screen "04_Izleme" 800x480, template "MainTemplate"
   TextField "Text field_1" at 81,3 size 108x20; Text 'En Ayar Pistonu'
   TextField "Text field_2" at 139,27 size 51x20; Text 'İleride'
   Circle "Circle_1" at 148,52 size 34x34
      Appearance <- "Peripheral_Data_IN_EnAyar_P1_Ileride"
   TextField "Text field_3" at 200,27 size 51x20; Text 'Geride'
   Circle "Circle_2" at 209,52 size 34x34
      Appearance <- "Peripheral_Data_IN_EnAyar_P1_Geride"
   Circle "Circle_3" at 148,96 size 34x34
      Appearance <- "Peripheral_Data_IN_EnAyar_P2_Ileride"
   Circle "Circle_4" at 209,96 size 34x34
      Appearance <- "Peripheral_Data_IN_EnAyar_P2_Geride"
   TextField "Text field_4" at 42,60 size 60x20; Text 'P1 (sol):'
   TextField "Text field_5" at 43,101 size 65x20; Text 'P2 (sağ):'
   Circle "Circle_5" at 148,138 size 34x34
      Appearance <- "Peripheral_Data_IN_EnAyar_P1A_Ileride"
   Circle "Circle_6" at 209,138 size 34x34
      Appearance <- "Peripheral_Data_IN_EnAyar_P1A_Geride"
   Circle "Circle_7" at 148,182 size 34x34
      Appearance <- "Peripheral_Data_IN_EnAyar_P2A_Ileride"
   Circle "Circle_8" at 209,182 size 34x34
      Appearance <- "Peripheral_Data_IN_EnAyar_P2A_Geride"
   TextField "Text field_6" at 42,146 size 70x20; Text 'P1A (sol):'
   TextField "Text field_7" at 43,187 size 75x20; Text 'P2A (sağ):'
   TextField "Text field_8" at 606,3 size 108x20; Text 'Kademe Pistonu'
   TextField "Text field_9" at 664,27 size 51x20; Text 'İleride'
   Circle "Circle_9" at 673,52 size 34x34
      Appearance <- "Peripheral_Data_IN_KademeAyar_P3_Ileride"
   TextField "Text field_10" at 725,27 size 51x20; Text 'Geride'
   Circle "Circle_10" at 734,52 size 34x34
      Appearance <- "Peripheral_Data_IN_KademeAyar_P3_Geride"
   TextField "Text field_11" at 567,60 size 26x20; Text 'P3:'
   TextField "Text field_13" at 318,2 size 155x20; Text 'Kenetleme Pistonu'
   TextField "Text field_14" at 401,26 size 51x20; Text 'İleride'
   Circle "Circle_13" at 410,51 size 34x34
      Appearance <- "Peripheral_Data_IN_Kenetleme_P4_Ilderide"
   TextField "Text field_15" at 462,26 size 51x20; Text 'Geride'
   Circle "Circle_14" at 471,51 size 34x34
      Appearance <- "Peripheral_Data_IN_Kenetleme_P4_Geride"
   TextField "Text field_16" at 304,59 size 65x20; Text 'P4 (sağ):'
   Circle "Circle_17" at 410,96 size 34x34
      Appearance <- "Peripheral_Data_IN_Kenetleme_P4B_Ilderide"
   Circle "Circle_18" at 471,96 size 34x34
      Appearance <- "Peripheral_Data_IN_Kenetleme_P4B_Geride"
   TextField "Text field_18" at 304,104 size 68x20; Text 'P4B (sol):'
   TextField "Text field_20" at 81,231 size 108x20; Text 'İkaz Lambaları'
   Circle "Circle_21" at 178,260 size 34x34
      Appearance <- "Peripheral_Data_OUT_LAMBA_Yesil"
   TextField "Text field_23" at 42,268 size 40x20; Text 'Yeşil:'
   TextField "Text field_21" at 322,231 size 155x20; Text 'Diğer Ekipmanlar'
   Circle "Circle_22" at 441,261 size 34x34
      Appearance <- "Peripheral_Data_OUT_VacumJeneratoru"
   TextField "Text field_22" at 304,268 size 53x20; Text 'Vakum:'
   Circle "Circle_24" at 441,305 size 34x34
      Appearance <- "Peripheral_Data_OUT_VincLambasi"
   TextField "Text field_25" at 304,311 size 93x20; Text 'Vinc Lambası:'
   Circle "Circle_25" at 177,305 size 34x34
      Appearance <- "Peripheral_Data.OUT.LAMBA.Sari"
   TextField "Text field_26" at 42,310 size 35x20; Text 'Sarı:'
   Circle "Circle_11" at 440,351 size 34x34
      Appearance <- "Peripheral_Data.OUT.LAMBA.Buzzer"
   TextField "Text field_12" at 305,356 size 43x20; Text 'Siren:'
   Circle "Circle_23" at 178,351 size 34x34
      Appearance <- "Peripheral_Data_OUT_LAMBA_Kirmizi"
   TextField "Text field_24" at 43,356 size 51x20; Text 'Kırmızı:'
   TextField "Text field_17" at 149,59 size 30x20; Text 'I0.4'
   TextField "Text field_19" at 212,59 size 30x20; Text 'I0.5'
   TextField "Text field_27" at 149,103 size 30x20; Text 'I1.0'
   TextField "Text field_28" at 212,103 size 30x20; Text 'I1.1'
   TextField "Text field_29" at 149,145 size 30x20; Text 'I0.6'
   TextField "Text field_30" at 212,145 size 30x20; Text 'I0.7'
   TextField "Text field_31" at 149,189 size 30x20; Text 'I1.2'
   TextField "Text field_32" at 212,189 size 30x20; Text 'I1.3'
   TextField "Text field_33" at 411,57 size 30x20; Text 'I2.0'
   TextField "Text field_34" at 474,57 size 30x20; Text 'I2.1'
   TextField "Text field_35" at 412,102 size 30x20; Text 'I2.2'
   TextField "Text field_36" at 474,102 size 30x20; Text 'I2.3'
   TextField "Text field_37" at 674,59 size 30x20; Text 'I1.4'
   TextField "Text field_38" at 737,59 size 30x20; Text 'I1.5'
   TextField "Text field_39" at 178,267 size 34x20; Text 'Q0.2'
   TextField "Text field_40" at 178,311 size 34x20; Text 'Q0.1'
   TextField "Text field_41" at 178,357 size 34x20; Text 'Q0.0'
   TextField "Text field_42" at 440,267 size 34x20; Text 'Q0.3'
   TextField "Text field_43" at 440,310 size 34x20; Text 'Q0.4'
   TextField "Text field_44" at 440,357 size 34x20; Text 'Q0.5'

screen "05_Receipt" 800x480, template "MainTemplate"
   TextField "Text field_1" at 258,159 size 300x124; Text 'KAYDEDİLDİ'
      Visibility <- "Receipt_bShowMessage"
   TextField "Template_Text field_1" at 45,17 size 109x22; Text 'Model Seçimi:'
   SymbolicIOField "Template_Symbolic I/O field_1" at 270,13 size 524x32; TextOn '1'; TextOff '0'; TextList "textListReceipt"
      ProcessValue <- "ModelId"
   Button "btnSave" at 619,337 size 167x58; TextOff 'KAYDET'
      on Release: SetBit("Receipt_btnSave")
   TextField "Template_Text field_4" at 45,139 size 124x22; Text 'Model Boyu (C):'
   TextField "Template_Text field_2" at 46,57 size 83x22; Text 'Model Adı:'
   IOField "I/O field_1" at 274,53 size 524x32; FormatPattern ??????????????????????????????????????????????????
      ProcessValue <- "ModelName"
   IOField "I/O field_2" at 273,134 size 256x32; FormatPattern s9999999.99; Unit  mm
      ProcessValue <- "Receipt_CurrentModel_Boy_C"
   TextField "Template_Text field_5" at 46,181 size 111x22; Text 'Model Eni (D):'
   IOField "I/O field_3" at 274,175 size 256x32; FormatPattern s9999999.99; Unit  mm
      ProcessValue <- "Receipt_CurrentModel_En_D"
   TextField "Template_Text field_3" at 45,98 size 99x22; Text 'Model Sınıfı:'
   SymbolicIOField "Template_Symbolic I/O field_2" at 275,94 size 68x32; TextOn '1'; TextOff '0'; TextList "classList"
      ProcessValue <- "Receipt_CurrentModel_Class"
   IOField "I/O field_4" at 275,290 size 185x32; FormatPattern 99999.99; Unit  mm
      ProcessValue <- "HMI_Data_ServoData_txtGerdirmeMes"
   TextField "Template_Text field_6" at 46,294 size 151x22; Text 'Gerdirme Mesafesi:'
   TextField "Template_Text field_7" at 45,252 size 154x23; Text 'Kenetleme Süresi:'
   IOField "Template_I/O field_1" at 275,248 size 184x32; FormatPattern 9999999999; Unit  sn
      ProcessValue <- "HMI_Data_KenetlemeSuresi"

screen "06_Alarm" 800x480, template "MainTemplate"
   AlarmView "Alarm view_1" at 2,1 size 796x415

screen "Screen_1" 800x480
   TextField "Text field_4" at 293,58 size 227x20; Text 'SERVO OTOMATİK KONTROL'
   IOField "I/O field_4" at 304,101 size 202x39; FormatPattern 999.9; Unit  %
      ProcessValue <- "HMI_Data_ServoData_txtVelocity"
   TextField "Text field_6" at 74,110 size 134x20; Text 'OTOMATİK MOD HIZ:'
   Button "btnIncJogSpeedXaxis_1" at 224,102 size 74x37; TextOff '-'
      on Release: function_b9b71300("HMI_Data_ServoData_txtVelocity", 5)
   Button "Button_1" at 512,102 size 75x37; TextOff '+'
      on Release: function_dd21b452("HMI_Data_ServoData_txtVelocity", 5)
   Button "Button_2" at 289,340 size 222x55; TextOff 'START'
      on Press: function_b14e0dd5("btnStartForHmi", 0)
   Button "Button_7" at 286,228 size 214x55; TextOff 'Aktif / Pasif'
      on Release: InvertBit("HMI_Data.Buttons.btnVakumJeneratoru")
   Rectangle "Rectangle_17" at 502,228 size 13x55
      Appearance <- "Peripheral_Data_OUT_VacumJeneratoru"
   TextField "Text field_3" at 327,204 size 140x20; Text 'Vakum Jeneratoru'
*)